# B&R Automation Studio project A2019059_Linka_Power_CP (part 27)

```iecst
        290:
            SC_P2_StoperSrobovania.StepName:='290 - Automaticky Rezim - modwel 5F presun manipulatora vzad';
            SC_P2_StoperSrobovania.IdleTime.PT:= T#200ms;
            SC_P2_StoperSrobovania.AlarmTime.PT:= T#5s;

            IF NOT SC_P2_StoperSrobovania.Switch1 AND P2_Robot.KOM_IN.Stav_RobotBezpPozicia_Srobovanie THEN
                P2_StoperSrobovania.OUT.KOM_PresunManipulator_DOZADU:= TRUE;
                SC_P2_StoperSrobovania.Switch1:= TRUE;
            END_IF

            IF P2_Srobovanie.OUT.KOM_PresunVZAD_Ukonceny THEN
                P2_Srobovanie.OUT.KOM_PresunVZAD_Ukonceny:= FALSE;
                P2_StoperSrobovania.OUT.KOM_PresunManipulator_DOZADU:= FALSE;
                CAM10.STAV.Results_READY:= FALSE;
                SC_P2_StoperSrobovania.ResetStep:= TRUE;
                SC_P2_StoperSrobovania.Step:= 293;
            END_IF

        293:
            SC_P2_StoperSrobovania.StepName:='293 - Automaticky Rezim - modwel 5F kamerova kontrola paletky CAM10';//CAM 10//
            SC_P2_StoperSrobovania.IdleTime.PT:= T#5s;
            SC_P2_StoperSrobovania.AlarmTime.PT:= T#5s;

            IF NOT SC_P2_StoperSrobovania.Switch1 AND CAM10.STAV.Command_READY THEN
                CAM10.CMD.Triger:= TRUE;
                SC_P2_StoperSrobovania.IdleTime.IN:= TRUE;
                SC_P2_StoperSrobovania.Switch1:= TRUE;
            END_IF

            IF CAM10.STAV.Results_READY AND CAM10.STAV.Command_AKCEPTOVANY THEN
                PocetTrigrovKamery:= 0;
                CAM10.STAV.Results_READY:= FALSE;
                SC_P2_StoperSrobovania.ResetStep:= TRUE;
                SC_P2_StoperSrobovania.Step:= 295;
            ELSIF SC_P2_StoperSrobovania.IdleTime.Q AND PocetTrigrovKamery < 5 THEN
                PocetTrigrovKamery:= PocetTrigrovKamery + 1;
                CAM10.STAV.Results_READY:= FALSE;
                CAM10.CMD.Triger:= FALSE;
                SC_P2_StoperSrobovania.ResetStep:= TRUE;
                SC_P2_StoperSrobovania.Step:= 294;
            ELSIF SC_P2_StoperSrobovania.IdleTime.Q AND PocetTrigrovKamery >= 5 THEN
                P2_Alarmy[295]:= TRUE;
                P2_PoruchaST3:= TRUE;
            END_IF

        294:
            SC_P2_StoperSrobovania.StepName:='294 - Automaticky Rezim - modwel 5F cakam na opatovny triger kamery';//CAM 10//
            SC_P2_StoperSrobovania.IdleTime.PT:= T#1s;
            SC_P2_StoperSrobovania.AlarmTime.PT:= T#5s;

            SC_P2_StoperSrobovania.IdleTime.IN:= TRUE;

            IF SC_P2_StoperSrobovania.IdleTime.Q THEN
                SC_P2_StoperSrobovania.ResetStep:= TRUE;
                SC_P2_StoperSrobovania.Step:= 293;
            END_IF

        295:
            SC_P2_StoperSrobovania.StepName:='295 - Automaticky Rezim - model 5F kontrola vysledku kamery';
            SC_P2_StoperSrobovania.IdleTime.PT:= T#200ms;
            SC_P2_StoperSrobovania.AlarmTime.PT:= T#5s;
            SC_P2_StoperSrobovania.IdleTime.IN:= TRUE;

            IF NOT CAM10.STAV.BUSY THEN
                CAM10.CMD.Triger:= FALSE;
				IF NOT CAM10.RESULT.Paletka.Pritomn_Busbarov_5F THEN
					CAM10.PAR.ResultFotky:= 'PASS';
					SC_P2_StoperSrobovania.ResetStep:= TRUE;
					SC_P2_StoperSrobovania.Step:= 300;
				ELSE
                    CAM10.PAR.ResultFotky:= 'FAIL';
                    SC_P2_StoperSrobovania.ResetStep:= TRUE;
                    SC_P2_StoperSrobovania.Step:= 300;
                END_IF
            END_IF

        300:
            SC_P2_StoperSrobovania.StepName:='300 - Automaticky Rezim - model 5F rozhodnutie podla kamerovej kontroly paletky';
            SC_P2_StoperSrobovania.IdleTime.PT:= T#200ms;
            SC_P2_StoperSrobovania.AlarmTime.PT:= T#5s;
            P2_Srobov_CakaNaKameru:= TRUE;

            IF CAM10.PAR.ResultFotky = 'PASS' THEN
                Paletka[i].PAR.StavPowerCP:= 'PASS';
                Paletka[i].VnutornyStav.CinnostUkoncena:= TRUE;
                P2_Srobov_CakaNaKameru:= FALSE;
                SC_P2_StoperSrobovania.ResetStep:= TRUE;
                SC_P2_StoperSrobovania.Step:= 540;
            ELSIF CAM10.PAR.ResultFotky = 'FAIL' THEN
                P2_Vizu.ZobrazHL2_ST5:= TRUE;
                Paletka[i].VnutornyStav.CinnostUkoncena:= TRUE;
                IF P2_Srobov_KAM_Result_OFF THEN
                    Paletka[i].PAR.StavPowerCP:= 'PASS';
                    P2_Vizu.ZobrazHL2_ST5:= FALSE;
                    P2_Srobov_CakaNaKameru:= FALSE;
                    SC_P2_StoperSrobovania.ResetStep:= TRUE;
                    SC_P2_StoperSrobovania.Step:= 540;
                ELSIF P2_Srobov_KAM_Result_OK THEN
                    P2_Srobov_KAM_Result_OK:= FALSE;
                    Paletka[i].PAR.StavPowerCP:= 'PASS';
                    CAM10.PAR.ResultFotky:= 'PASS';
                    P2_Srobov_CakaNaKameru:= FALSE;
                    P2_Vizu.ZobrazHL2_ST5:= FALSE;
                    SC_P2_StoperSrobovania.ResetStep:= TRUE;
                    SC_P2_StoperSrobovania.Step:= 540;
                ELSIF P2_Srobov_KAM_Result_NG THEN
                    P2_Srobov_KAM_Result_NG:= FALSE;
                    P2_Vizu.ZobrazHL2_ST5:= FALSE;
                    Paletka[i].PAR.StavPowerCP:= 'FAIL';
                    P2_Srobov_CakaNaKameru:= FALSE;
                    SC_P2_StoperSrobovania.ResetStep:= TRUE;
                    SC_P2_StoperSrobovania.Step:= 540;
                END_IF
            END_IF

            //********************************************Model 5H**************************************************************//

        358:
            SC_P2_StoperSrobovania.StepName:='358 - Automaticky Rezim - model 5H presun manipulatora vpred a odobratie vrchnych busbarov';
            SC_P2_StoperSrobovania.IdleTime.PT:= T#200ms;
            SC_P2_StoperSrobovania.AlarmTime.PT:= T#5s;

            P2_Robot.KOM_OUT.ManipSrobovania_BezpecnaPozicia:= TRUE;

            IF P2_Robot.KOM_IN.Stav_RobotBezpPozicia_Srobovanie AND NOT P2_Robot.KOM_IN.Stav_Busbary5H_Odobrate AND NOT P2_Robot.STAV.Zvaranie_PrebiehaManipulacia AND SC_P2_Srobovanie.Step = 100  THEN
                P2_StoperSrobovania.OUT.KOM_PresunManipulator_DOPREDU:= TRUE;
                P2_Robot.KOM_OUT.Odober_Busbary5H:= TRUE;
                Paletka[i].VnutornyStav.CinnostSpustena:= TRUE;
                SC_P2_StoperSrobovania.ResetStep:= TRUE;
                SC_P2_StoperSrobovania.Step:= 360;
            ELSIF NOT P2_Robot.KOM_IN.Stav_ProgramRUN THEN
                P2_Alarmy[271]:= TRUE;
                P2_PoruchaST3:= TRUE;
            END_IF

        360:
            SC_P2_StoperSrobovania.StepName:='360 - Automaticky Rezim - modwel 5H cakam na polozenie vrchnych busbarov';
            SC_P2_StoperSrobovania.IdleTime.PT:= T#200ms;
            SC_P2_StoperSrobovania.AlarmTime.PT:= T#5s;

            IF P2_Srobovanie.OUT.KOM_PresunVPRED_Ukonceny AND P2_Robot.KOM_IN.Stav_Busbary5H_Odobrate AND NOT P2_Robot.KOM_IN.Stav_Busbary5H_Polozene THEN
                P2_Srobovanie.OUT.KOM_PresunVPRED_Ukonceny:= FALSE;
                P2_StoperSrobovania.OUT.KOM_PresunManipulator_DOPREDU:= FALSE;
                P2_Robot.KOM_OUT.Odober_Busbary5H:= FALSE;
                SC_P2_StoperSrobovania.ResetStep:= TRUE;
                SC_P2_StoperSrobovania.Step:= 363;
            ELSIF NOT P2_Robot.KOM_IN.Stav_ProgramRUN THEN
                P2_Alarmy[271]:= TRUE;
                P2_PoruchaST3:= TRUE;
            END_IF

        363:
            SC_P2_StoperSrobovania.StepName:='363 - Automaticky Rezim - modwel 5H poloz vrchne busbary';
            SC_P2_StoperSrobovania.IdleTime.PT:= T#200ms;
            SC_P2_StoperSrobovania.AlarmTime.PT:= T#5s;

            P2_Robot.KOM_OUT.ManipSrobovania_BezpecnaPozicia:= TRUE;

            IF NOT SC_P2_StoperSrobovania.Switch1 AND NOT P2_Robot.KOM_IN.Stav_Busbary5H_Odobrate THEN
                P2_Robot.KOM_OUT.Poloz_Busbary5H:= TRUE;
                SC_P2_StoperSrobovania.Switch1:= TRUE;
            END_IF

            IF P2_Robot.KOM_IN.Stav_Busbary5H_Polozene THEN
                P2_Robot.KOM_OUT.Poloz_Busbary5H:= FALSE;
                SC_P2_StoperSrobovania.ResetStep:= TRUE;
                SC_P2_StoperSrobovania.Step:= 365;
            ELSIF NOT P2_Robot.KOM_IN.Stav_ProgramRUN THEN
                P2_Alarmy[271]:= TRUE;
                P2_PoruchaST3:= TRUE;
            END_IF

        365:
            SC_P2_StoperSrobovania.StepName:='365 - Automaticky Rezim - modwel 5H zaskrutkuj skrutku M4';
            SC_P2_StoperSrobovania.IdleTime.PT:= T#200ms;
            SC_P2_StoperSrobovania.AlarmTime.PT:= T#5s;

            IF NOT SC_P2_StoperSrobovania.Switch1 THEN
                P2_Srobovanie.STAV.Vysledok_Srobovania:= '';
                P2_StoperSrobovania.OUT.KOM_5H_ZasrobujSkrutkuM4:= TRUE;
                SC_P2_StoperSrobovania.Switch1:= TRUE;
            END_IF

            IF P2_Srobovanie.OUT.KOM_Srobovanie_Ukoncene AND NOT P2_Robot.KOM_IN.Stav_Filter5H_Dotlaceny THEN
                P2_Srobovanie.OUT.KOM_Srobovanie_Ukoncene:= FALSE;
                P2_StoperSrobovania.OUT.KOM_5H_ZasrobujSkrutkuM4:= FALSE;
                IF P2_StoperSrobovania.STAV.Porucha THEN
                    SC_P2_StoperSrobovania.ResetStep:= TRUE;
                    SC_P2_StoperSrobovania.Step:= 500;//500
                ELSE
                    SC_P2_StoperSrobovania.ResetStep:= TRUE;
                    SC_P2_StoperSrobovania.Step:= 368;
                END_IF
            END_IF

        368:
            SC_P2_StoperSrobovania.StepName:='368 - Automaticky Rezim - modwel 5H kontrola vysledku zaskrutkovania skrutky M4';
            SC_P2_StoperSrobovania.IdleTime.PT:= T#200ms;
            SC_P2_StoperSrobovania.AlarmTime.PT:= T#5s;

            Reports.Skrutkovacky.Moment_ToleranciaMIN.P2_StrednaSkrutkaM4:= REAL_TO_STRING(P2_Srobovanie.STAV.M4_Moment_ToleranciaMIN_REAL);
            Reports.Skrutkovacky.Moment_ToleranciaMAX.P2_StrednaSkrutkaM4:= REAL_TO_STRING(P2_Srobovanie.STAV.M4_Moment_ToleranciaMAX_REAL);
            Reports.Skrutkovacky.Moment_NameranaHodnota.P2_StrednaSkrutkaM4:= REAL_TO_STRING(P2_Srobovanie.STAV.M4_DosiahnutyMoment_REAL);
            Reports.Skrutkovacky.Uhol_ToleranciaMIN.P2_StrednaSkrutkaM4:= UDINT_TO_STRING(P2_Srobovanie.STAV.M4_Uhol_ToleranciaMIN);
            Reports.Skrutkovacky.Uhol_ToleranciaMAX.P2_StrednaSkrutkaM4:= UDINT_TO_STRING(P2_Srobovanie.STAV.M4_Uhol_ToleranciaMAX);
            Reports.Skrutkovacky.Uhol_NameranaHodnota.P2_StrednaSkrutkaM4:= UDINT_TO_STRING(P2_Srobovanie.STAV.M4_DosiahnutyUhol);

            IF NOT SC_P2_StoperSrobovania.Switch1 THEN
                P2_Skrutk_5H_StrednaM4_Vysunutie:= STRING_TO_REAL(Reports.Skrutkovacky.VyskaSkrutkovania.P2_StrednaSkrutkaM4);
                IF (P2_Skrutk_5H_StrednaM4_Vysunutie <= P2_RemPremenne.P2_Srob5H_StrednaM4_Vysunutie_HI) AND (P2_Skrutk_5H_StrednaM4_Vysunutie >= P2_RemPremenne.P2_Srob5H_StrednaM4_Vysunutie_LO)THEN
                    VysunutieSkrutkovacky_OK:= TRUE;
                ELSE
                    VysunutieSkrutkovacky_OK:= FALSE;
                END_IF
                SC_P2_StoperSrobovania.Switch1:= TRUE;
            END_IF

            IF P2_Srobovanie.STAV.Vysledok_Srobovania = 'OK' THEN
                IF VysunutieSkrutkovacky_OK THEN
                    Reports.Skrutkovacky.VyslednyReport.P2_StrednaSkrutkaM4:= 'PASS';
                    SC_P2_StoperSrobovania.ResetStep:= TRUE;
                    SC_P2_StoperSrobovania.Step:= 370;
                ELSE
                    Reports.Skrutkovacky.VyslednyReport.P2_StrednaSkrutkaM4:= 'FAIL';
                    IF P2_Srobov_M4_Result_OFF THEN
                        SC_P2_StoperSrobovania.ResetStep:= TRUE;
                        SC_P2_StoperSrobovania.Step:= 370;
                    ELSE
                        DoskrutkovaniePriPoruche:= TRUE;
                        SC_P2_StoperSrobovania.ResetStep:= TRUE;
                        SC_P2_StoperSrobovania.Step:= 370;//500
                    END_IF
                END_IF
            ELSIF P2_Srobovanie.STAV.Vysledok_Srobovania = 'NG' THEN
                Reports.Skrutkovacky.VyslednyReport.P2_StrednaSkrutkaM4:= 'FAIL';
                IF P2_Srobov_M4_Result_OFF THEN
                    SC_P2_StoperSrobovania.ResetStep:= TRUE;
                    SC_P2_StoperSrobovania.Step:= 370;
                ELSE
                    DoskrutkovaniePriPoruche:= TRUE;
                    SC_P2_StoperSrobovania.ResetStep:= TRUE;
                    SC_P2_StoperSrobovania.Step:= 370;//500
                END_IF
            END_IF

        370:
            SC_P2_StoperSrobovania.StepName:='370 - Automaticky Rezim - modwel 5H dotlac filter';
            SC_P2_StoperSrobovania.IdleTime.PT:= T#200ms;
            SC_P2_StoperSrobovania.AlarmTime.PT:= T#5s;

            P2_Robot.KOM_OUT.ManipSrobovania_BezpecnaPozicia:= TRUE;

            IF NOT SC_P2_StoperSrobovania.Switch1 THEN
                P2_Robot.KOM_OUT.Dotlac_Filter5H:= TRUE;
                SC_P2_StoperSrobovania.Switch1:= TRUE;
            END_IF

            IF P2_Robot.KOM_IN.Stav_Filter5H_Dotlaceny THEN
                P2_Robot.KOM_OUT.Dotlac_Filter5H:= FALSE;
                SC_P2_StoperSrobovania.ResetStep:= TRUE;
                SC_P2_StoperSrobovania.Step:= 375;
            ELSIF NOT P2_Robot.KOM_IN.Stav_ProgramRUN THEN
                P2_Alarmy[271]:= TRUE;
                P2_PoruchaST3:= TRUE;
            END_IF

        375:
            SC_P2_StoperSrobovania.StepName:='375 - Automaticky Rezim - modwel 5H zaskrutkuj lavu skrutku M5';
            SC_P2_StoperSrobovania.IdleTime.PT:= T#200ms;
            SC_P2_StoperSrobovania.AlarmTime.PT:= T#5s;

            IF NOT SC_P2_StoperSrobovania.Switch1 THEN
                P2_Srobovanie.STAV.Vysledok_Srobovania:= '';
                P2_StoperSrobovania.OUT.KOM_5H_ZasrobujLavuSkrutkuM5:= TRUE;
                SC_P2_StoperSrobovania.Switch1:= TRUE;
            END_IF

            IF P2_Srobovanie.OUT.KOM_Srobovanie_Ukoncene THEN
                P2_Srobovanie.OUT.KOM_Srobovanie_Ukoncene:= FALSE;
                P2_StoperSrobovania.OUT.KOM_5H_ZasrobujLavuSkrutkuM5:= FALSE;
                IF P2_StoperSrobovania.STAV.Porucha THEN
                    SC_P2_StoperSrobovania.ResetStep:= TRUE;
                    SC_P2_StoperSrobovania.Step:= 500;
                ELSE
                    SC_P2_StoperSrobovania.ResetStep:= TRUE;
                    SC_P2_StoperSrobovania.Step:= 378;
                END_IF
            END_IF

        378:
            SC_P2_StoperSrobovania.StepName:='378 - Automaticky Rezim - modwel 5H kontrola vysledku zaskrutkovania lavej skrutky M5';
            SC_P2_StoperSrobovania.IdleTime.PT:= T#200ms;
            SC_P2_StoperSrobovania.AlarmTime.PT:= T#5s;

            Reports.Skrutkovacky.Moment_ToleranciaMIN.P2_LavaSkrutkaM5:= REAL_TO_STRING(P2_Srobovanie.STAV.M5_Moment_ToleranciaMIN_REAL);
            Reports.Skrutkovacky.Moment_ToleranciaMAX.P2_LavaSkrutkaM5:= REAL_TO_STRING(P2_Srobovanie.STAV.M5_Moment_ToleranciaMAX_REAL);
            Reports.Skrutkovacky.Moment_NameranaHodnota.P2_LavaSkrutkaM5:= REAL_TO_STRING(P2_Srobovanie.STAV.M5_DosiahnutyMoment_REAL);
            Reports.Skrutkovacky.Uhol_ToleranciaMIN.P2_LavaSkrutkaM5:= UDINT_TO_STRING(P2_Srobovanie.STAV.M5_Uhol_ToleranciaMIN);
            Reports.Skrutkovacky.Uhol_ToleranciaMAX.P2_LavaSkrutkaM5:= UDINT_TO_STRING(P2_Srobovanie.STAV.M5_Uhol_ToleranciaMAX);
            Reports.Skrutkovacky.Uhol_NameranaHodnota.P2_LavaSkrutkaM5:= UDINT_TO_STRING(P2_Srobovanie.STAV.M5_DosiahnutyUhol);

            IF NOT SC_P2_StoperSrobovania.Switch1 THEN
                P2_Skrutk_5H_LavaM5_Vysunutie:= STRING_TO_REAL(Reports.Skrutkovacky.VyskaSkrutkovania.P2_LavaSkrutkaM5);
                IF (P2_Skrutk_5H_LavaM5_Vysunutie <= P2_RemPremenne.P2_Srob5H_LavaM5_Vysunutie_HI) AND (P2_Skrutk_5H_LavaM5_Vysunutie >= P2_RemPremenne.P2_Srob5H_LavaM5_Vysunutie_LO)THEN
                    VysunutieSkrutkovacky_OK:= TRUE;
                ELSE
                    VysunutieSkrutkovacky_OK:= FALSE;
                END_IF
                SC_P2_StoperSrobovania.Switch1:= TRUE;
            END_IF

            IF P2_Srobovanie.STAV.Vysledok_Srobovania = 'OK' THEN
                IF VysunutieSkrutkovacky_OK THEN
                    IF NOT DoskrutkovaniePriPoruche THEN
                        Reports.Skrutkovacky.VyslednyReport.P2_LavaSkrutkaM5:= 'PASS';
                    ELSE
                        Reports.Skrutkovacky.VyslednyReport.P2_LavaSkrutkaM5:= 'FAIL';
                    END_IF
                    SC_P2_StoperSrobovania.ResetStep:= TRUE;
                    SC_P2_StoperSrobovania.Step:= 380;
                ELSE
                    Reports.Skrutkovacky.VyslednyReport.P2_LavaSkrutkaM5:= 'FAIL';
                    IF P2_Srobov_M5_Result_OFF THEN
                        SC_P2_StoperSrobovania.ResetStep:= TRUE;
                        SC_P2_StoperSrobovania.Step:= 380;
                    ELSE
                        DoskrutkovaniePriPoruche:= TRUE;
                        SC_P2_StoperSrobovania.ResetStep:= TRUE;
                        SC_P2_StoperSrobovania.Step:= 380;//500
                    END_IF
                END_IF
            ELSIF P2_Srobovanie.STAV.Vysledok_Srobovania = 'NG' THEN
                Reports.Skrutkovacky.VyslednyReport.P2_LavaSkrutkaM5:= 'FAIL';
                IF P2_Srobov_M5_Result_OFF THEN
                    SC_P2_StoperSrobovania.ResetStep:= TRUE;
                    SC_P2_StoperSrobovania.Step:= 380;
                ELSE
                    DoskrutkovaniePriPoruche:= TRUE;
                    SC_P2_StoperSrobovania.ResetStep:= TRUE;
                    SC_P2_StoperSrobovania.Step:= 380;//500
                END_IF
            END_IF

        380:
            SC_P2_StoperSrobovania.StepName:='380 - Automaticky Rezim - modwel 5H zaskrutkuj pravu skrutku M5';
            SC_P2_StoperSrobovania.IdleTime.PT:= T#200ms;
            SC_P2_StoperSrobovania.AlarmTime.PT:= T#5s;

            IF NOT SC_P2_StoperSrobovania.Switch1  THEN
                P2_Srobovanie.STAV.Vysledok_Srobovania:= '';
                P2_StoperSrobovania.OUT.KOM_5H_ZasrobujPravuSkrutkuM5:= TRUE;
                SC_P2_StoperSrobovania.Switch1:= TRUE;
            END_IF

            IF P2_Srobovanie.OUT.KOM_Srobovanie_Ukoncene THEN
                P2_Srobovanie.OUT.KOM_Srobovanie_Ukoncene:= FALSE;
                P2_StoperSrobovania.OUT.KOM_5H_ZasrobujPravuSkrutkuM5:= FALSE;
                IF P2_StoperSrobovania.STAV.Porucha THEN
                    SC_P2_StoperSrobovania.ResetStep:= TRUE;
                    SC_P2_StoperSrobovania.Step:= 500;
                ELSE
                    SC_P2_StoperSrobovania.ResetStep:= TRUE;
                    SC_P2_StoperSrobovania.Step:= 383;
                END_IF
            END_IF

        383:
            SC_P2_StoperSrobovania.StepName:='383 - Automaticky Rezim - modwel 5H kontrola vysledku zaskrutkovania pravej skrutky M5';
            SC_P2_StoperSrobovania.IdleTime.PT:= T#200ms;
            SC_P2_StoperSrobovania.AlarmTime.PT:= T#5s;

            Reports.Skrutkovacky.Moment_ToleranciaMIN.P2_PravaSkrutkaM5:= REAL_TO_STRING(P2_Srobovanie.STAV.M5_Moment_ToleranciaMIN_REAL);
            Reports.Skrutkovacky.Moment_ToleranciaMAX.P2_PravaSkrutkaM5:= REAL_TO_STRING(P2_Srobovanie.STAV.M5_Moment_ToleranciaMAX_REAL);
            Reports.Skrutkovacky.Moment_NameranaHodnota.P2_PravaSkrutkaM5:= REAL_TO_STRING(P2_Srobovanie.STAV.M5_DosiahnutyMoment_REAL);
            Reports.Skrutkovacky.Uhol_ToleranciaMIN.P2_PravaSkrutkaM5:= UDINT_TO_STRING(P2_Srobovanie.STAV.M5_Uhol_ToleranciaMIN);
            Reports.Skrutkovacky.Uhol_ToleranciaMAX.P2_PravaSkrutkaM5:= UDINT_TO_STRING(P2_Srobovanie.STAV.M5_Uhol_ToleranciaMAX);
            Reports.Skrutkovacky.Uhol_NameranaHodnota.P2_PravaSkrutkaM5:= UDINT_TO_STRING(P2_Srobovanie.STAV.M5_DosiahnutyUhol);

            IF NOT SC_P2_StoperSrobovania.Switch1 THEN
                P2_Skrutk_5H_PravaM5_Vysunutie:= STRING_TO_REAL(Reports.Skrutkovacky.VyskaSkrutkovania.P2_PravaSkrutkaM5);
                IF (P2_Skrutk_5H_PravaM5_Vysunutie <= P2_RemPremenne.P2_Srob5H_PravaM5_Vysunutie_HI) AND (P2_Skrutk_5H_PravaM5_Vysunutie >= P2_RemPremenne.P2_Srob5H_PravaM5_Vysunutie_LO)THEN
                    VysunutieSkrutkovacky_OK:= TRUE;
                ELSE
                    VysunutieSkrutkovacky_OK:= FALSE;
                END_IF
                SC_P2_StoperSrobovania.Switch1:= TRUE;
            END_IF

            IF P2_Srobovanie.STAV.Vysledok_Srobovania = 'OK' THEN
                IF VysunutieSkrutkovacky_OK THEN
                    IF NOT DoskrutkovaniePriPoruche THEN
                        Reports.Skrutkovacky.VyslednyReport.P2_PravaSkrutkaM5:= 'PASS';
                        SC_P2_StoperSrobovania.ResetStep:= TRUE;
                        SC_P2_StoperSrobovania.Step:= 385;
                    ELSE
                        Reports.Skrutkovacky.VyslednyReport.P2_PravaSkrutkaM5:= 'FAIL';
                        SC_P2_StoperSrobovania.ResetStep:= TRUE;
                        SC_P2_StoperSrobovania.Step:= 500;
                    END_IF
                ELSE
                    Reports.Skrutkovacky.VyslednyReport.P2_PravaSkrutkaM5:= 'FAIL';
                    IF P2_Srobov_M5_Result_OFF THEN
                        SC_P2_StoperSrobovania.ResetStep:= TRUE;
                        SC_P2_StoperSrobovania.Step:= 385;
                    ELSE
                        SC_P2_StoperSrobovania.ResetStep:= TRUE;
                        SC_P2_StoperSrobovania.Step:= 500;
                    END_IF
                END_IF
            ELSIF P2_Srobovanie.STAV.Vysledok_Srobovania = 'NG' THEN
                Reports.Skrutkovacky.VyslednyReport.P2_PravaSkrutkaM5:= 'FAIL';
                IF P2_Srobov_M5_Result_OFF THEN
                    SC_P2_StoperSrobovania.ResetStep:= TRUE;
                    SC_P2_StoperSrobovania.Step:= 385;
                ELSE
                    SC_P2_StoperSrobovania.ResetStep:= TRUE;
                    SC_P2_StoperSrobovania.Step:= 500;
                END_IF
            END_IF

        385:
            SC_P2_StoperSrobovania.StepName:='385 - Automaticky Rezim - modwel 5H presun manipulatora vpred, vystavenie signalu pre robota chod do cakacej pozicie ';
            SC_P2_StoperSrobovania.IdleTime.PT:= T#200ms;
            SC_P2_StoperSrobovania.AlarmTime.PT:= T#5s;

            P2_Robot.KOM_OUT.ManipSrobovania_BezpecnaPozicia:= TRUE;

            IF NOT P2_Robot.KOM_IN.Stav_RobotPoziciaCakania THEN
                P2_StoperSrobovania.OUT.KOM_PresunManipulator_DOPREDU:= TRUE;
                P2_Robot.KOM_OUT.Presun_CakaciaPozicia:= TRUE;
                SC_P2_StoperSrobovania.ResetStep:= TRUE;
                SC_P2_StoperSrobovania.Step:= 388;
            END_IF

        388:
            SC_P2_StoperSrobovania.StepName:='388 - Automaticky Rezim - model 5H cakam na presunutie robota do cakacej pozicie';
            SC_P2_StoperSrobovania.IdleTime.PT:= T#200ms;
            SC_P2_StoperSrobovania.AlarmTime.PT:= T#5s;

            IF P2_Srobovanie.OUT.KOM_PresunVPRED_Ukonceny AND P2_Robot.KOM_IN.Stav_RobotPoziciaCakania THEN
                P2_Robot.KOM_OUT.Presun_CakaciaPozicia:= FALSE;
                P2_Robot.STAV.Srobovanie_PrebiehaManipulacia:= FALSE;
                P2_Srobovanie.OUT.KOM_PresunVPRED_Ukonceny:= FALSE;
                P2_StoperSrobovania.OUT.KOM_PresunManipulator_DOPREDU:= FALSE;
                SC_P2_StoperSrobovania.ResetStep:= TRUE;
                SC_P2_StoperSrobovania.Step:= 390;
            END_IF

        390:
            SC_P2_StoperSrobovania.StepName:='390 - Automaticky Rezim - modwel 5H presun manipulatora vzad';
            SC_P2_StoperSrobovania.IdleTime.PT:= T#200ms;
            SC_P2_StoperSrobovania.AlarmTime.PT:= T#5s;

            IF NOT SC_P2_StoperSrobovania.Switch1 AND P2_Robot.KOM_IN.Stav_RobotBezpPozicia_Srobovanie AND SC_P2_Srobovanie.Step = 100 THEN
                P2_StoperSrobovania.OUT.KOM_PresunManipulator_DOZADU:= TRUE;
                SC_P2_StoperSrobovania.Switch1:= TRUE;
            END_IF

            IF P2_Srobovanie.OUT.KOM_PresunVZAD_Ukonceny THEN
                P2_Srobovanie.OUT.KOM_PresunVZAD_Ukonceny:= FALSE;
                P2_StoperSrobovania.OUT.KOM_PresunManipulator_DOZADU:= FALSE;
                CAM10.STAV.Results_READY:= FALSE;
                SC_P2_StoperSrobovania.ResetStep:= TRUE;
                SC_P2_StoperSrobovania.Step:= 393;
            END_IF

        393:
            SC_P2_StoperSrobovania.StepName:='393 - Automaticky Rezim - modwel 5H kamerova kontrola paletky CAM10';//CAM 10//
            SC_P2_StoperSrobovania.IdleTime.PT:= T#5s;
            SC_P2_StoperSrobovania.AlarmTime.PT:= T#5s;

            IF NOT SC_P2_StoperSrobovania.Switch1 AND CAM10.STAV.Command_READY THEN
                CAM10.CMD.Triger:= TRUE;
                SC_P2_StoperSrobovania.IdleTime.IN:= TRUE;
                SC_P2_StoperSrobovania.Switch1:= TRUE;
            END_IF

            IF CAM10.STAV.Results_READY AND CAM10.STAV.Command_AKCEPTOVANY THEN
                PocetTrigrovKamery:= 0;
                CAM10.STAV.Results_READY:= FALSE;
                SC_P2_StoperSrobovania.ResetStep:= TRUE;
                SC_P2_StoperSrobovania.Step:= 395;
            ELSIF SC_P2_StoperSrobovania.IdleTime.Q AND PocetTrigrovKamery < 5 THEN
                PocetTrigrovKamery:= PocetTrigrovKamery + 1;
                CAM10.STAV.Results_READY:= FALSE;
                CAM10.CMD.Triger:= FALSE;
                SC_P2_StoperSrobovania.ResetStep:= TRUE;
                SC_P2_StoperSrobovania.Step:= 394;
            ELSIF SC_P2_StoperSrobovania.IdleTime.Q AND PocetTrigrovKamery >= 5 THEN
                P2_Alarmy[295]:= TRUE;
                P2_PoruchaST3:= TRUE;
            END_IF

        394:
            SC_P2_StoperSrobovania.StepName:='394 - Automaticky Rezim - modwel 5H cakam na opatovny triger kamery';//CAM 10//
            SC_P2_StoperSrobovania.IdleTime.PT:= T#1s;
            SC_P2_StoperSrobovania.AlarmTime.PT:= T#5s;

            SC_P2_StoperSrobovania.IdleTime.IN:= TRUE;

            IF SC_P2_StoperSrobovania.IdleTime.Q THEN
                SC_P2_StoperSrobovania.ResetStep:= TRUE;
                SC_P2_StoperSrobovania.Step:= 393;
            END_IF

        395:
            SC_P2_StoperSrobovania.StepName:='395 - Automaticky Rezim - model 5H kontrola vysledku kamery';
            SC_P2_StoperSrobovania.IdleTime.PT:= T#200ms;
            SC_P2_StoperSrobovania.AlarmTime.PT:= T#5s;
            SC_P2_StoperSrobovania.IdleTime.IN:= TRUE;

            IF NOT CAM10.STAV.BUSY  THEN
                CAM10.CMD.Triger:= FALSE;
				IF NOT CAM10.RESULT.Paletka.Pritomn_Busbarov_5H THEN
					CAM10.PAR.ResultFotky:= 'PASS';
					SC_P2_StoperSrobovania.ResetStep:= TRUE;
					SC_P2_StoperSrobovania.Step:= 400;
                ELSE
                    CAM10.PAR.ResultFotky:= 'FAIL';
                    SC_P2_StoperSrobovania.ResetStep:= TRUE;
                    SC_P2_StoperSrobovania.Step:= 400;
                END_IF
            END_IF

        400:
            SC_P2_StoperSrobovania.StepName:='400 - Automaticky Rezim - model 5H rozhodnutie podla kamerovej kontroly paletky';
            SC_P2_StoperSrobovania.IdleTime.PT:= T#200ms;
            SC_P2_StoperSrobovania.AlarmTime.PT:= T#5s;
            P2_Srobov_CakaNaKameru:= TRUE;

            IF CAM10.PAR.ResultFotky = 'PASS' THEN
                Paletka[i].VnutornyStav.CinnostUkoncena:= TRUE;
                Paletka[i].PAR.StavPowerCP:= 'PASS';
                P2_Srobov_CakaNaKameru:= FALSE;
                SC_P2_StoperSrobovania.ResetStep:= TRUE;
                SC_P2_StoperSrobovania.Step:= 540;
            ELSIF CAM10.PAR.ResultFotky = 'FAIL' THEN
                P2_Vizu.ZobrazHL3_ST5:= TRUE;
                Paletka[i].VnutornyStav.CinnostUkoncena:= TRUE;
                IF P2_Srobov_KAM_Result_OFF THEN
                    Paletka[i].PAR.StavPowerCP:= 'PASS';
                    P2_Vizu.ZobrazHL3_ST5:= FALSE;
                    P2_Srobov_CakaNaKameru:= FALSE;
                    SC_P2_StoperSrobovania.ResetStep:= TRUE;
                    SC_P2_StoperSrobovania.Step:= 540;
                ELSIF P2_Srobov_KAM_Result_OK THEN
                    P2_Srobov_KAM_Result_OK:= FALSE;
                    Paletka[i].PAR.StavPowerCP:= 'PASS';
                    CAM10.PAR.ResultFotky:= 'PASS';
                    P2_Srobov_CakaNaKameru:= FALSE;
                    P2_Vizu.ZobrazHL3_ST5:= FALSE;
                    SC_P2_StoperSrobovania.ResetStep:= TRUE;
                    SC_P2_StoperSrobovania.Step:= 540;
                ELSIF P2_Srobov_KAM_Result_NG THEN
                    P2_Srobov_KAM_Result_NG:= FALSE;
                    P2_Vizu.ZobrazHL3_ST5:= FALSE;
                    Paletka[i].PAR.StavPowerCP:= 'FAIL';
                    P2_Srobov_CakaNaKameru:= FALSE;
                    SC_P2_StoperSrobovania.ResetStep:= TRUE;
                    SC_P2_StoperSrobovania.Step:= 540;
                END_IF
            END_IF

            //****************************************Uvolnenie robota a vyfotenie paletky po zlom skrutkovaní************************************************//

        500:
            SC_P2_StoperSrobovania.StepName:='500 - Automaticky Rezim - presun manipulatora vpred';
            SC_P2_StoperSrobovania.IdleTime.PT:= T#200ms;
            SC_P2_StoperSrobovania.AlarmTime.PT:= T#5s;

			Paletka[i].PAR.StavPaletky:= 'NG';

            IF NOT SC_P2_StoperSrobovania.Switch1 THEN
                P2_StoperSrobovania.OUT.KOM_PresunManipulator_DOPREDU:= TRUE;
                SC_P2_StoperSrobovania.Switch1:= TRUE;
            END_IF

            IF P2_Srobovanie.OUT.KOM_PresunVPRED_Ukonceny THEN
                P2_Srobovanie.OUT.KOM_PresunVPRED_Ukonceny:= FALSE;
                P2_StoperSrobovania.OUT.KOM_PresunManipulator_DOPREDU:= FALSE;
                SC_P2_StoperSrobovania.ResetStep:= TRUE;
                SC_P2_StoperSrobovania.Step:= 503;
            END_IF

        503:
            SC_P2_StoperSrobovania.StepName:='503 - Automaticky Rezim - vystavenie signalu pre robota chod do cakacej pozicie';
            SC_P2_StoperSrobovania.IdleTime.PT:= T#200ms;
            SC_P2_StoperSrobovania.AlarmTime.PT:= T#5s;

            P2_Robot.KOM_OUT.ManipSrobovania_BezpecnaPozicia:= TRUE;

            IF NOT SC_P2_StoperSrobovania.Switch1 THEN
                P2_Robot.KOM_OUT.Presun_CakaciaPozicia:= TRUE;
                SC_P2_StoperSrobovania.Switch1:= TRUE;
            END_IF

            IF P2_Robot.KOM_IN.Stav_RobotBezpPozicia_Srobovanie THEN
                P2_Robot.KOM_OUT.Presun_CakaciaPozicia:= FALSE;
                SC_P2_StoperSrobovania.ResetStep:= TRUE;
                SC_P2_StoperSrobovania.Step:= 505;
            END_IF

        505:
            SC_P2_StoperSrobovania.StepName:='505 - Automaticky Rezim - presun manipulatora vzad';
            SC_P2_StoperSrobovania.IdleTime.PT:= T#200ms;
            SC_P2_StoperSrobovania.AlarmTime.PT:= T#5s;

            IF NOT SC_P2_StoperSrobovania.Switch1 THEN
                P2_StoperSrobovania.OUT.KOM_PresunManipulator_DOZADU:= TRUE;
                SC_P2_StoperSrobovania.Switch1:= TRUE;
            END_IF

            IF P2_Srobovanie.OUT.KOM_PresunVZAD_Ukonceny THEN
                P2_Srobovanie.OUT.KOM_PresunVZAD_Ukonceny:= FALSE;
                P2_StoperSrobovania.OUT.KOM_PresunManipulator_DOZADU:= FALSE;
                IF P2_StoperSrobovania.STAV.Porucha THEN
                    CAM10.STAV.Results_READY:= FALSE;
                    SC_P2_StoperSrobovania.ResetStep:= TRUE;
                    SC_P2_StoperSrobovania.Step:= 545;
                ELSE
                    SC_P2_StoperSrobovania.ResetStep:= TRUE;
                    SC_P2_StoperSrobovania.Step:= 508;
                END_IF
            END_IF

        508:
            SC_P2_StoperSrobovania.StepName:='508 - Automaticky Rezim - kamerova kontrola paletky CAM10';//CAM 10//
            SC_P2_StoperSrobovania.IdleTime.PT:= T#5s;
            SC_P2_StoperSrobovania.AlarmTime.PT:= T#5s;
            SC_P2_StoperSrobovania.IdleTime.IN:= TRUE;

            IF NOT SC_P2_StoperSrobovania.Switch1 AND CAM10.STAV.Command_READY THEN
                CAM10.CMD.Triger:= TRUE;
                SC_P2_StoperSrobovania.Switch1:= TRUE;
            END_IF

            IF CAM10.STAV.Results_READY AND CAM10.STAV.Command_AKCEPTOVANY THEN
                PocetTrigrovKamery:= 0;
                CAM10.STAV.Results_READY:= FALSE;
                Paletka[i].PAR.StavPowerCP:= 'FAIL';
                CAM10.PAR.ResultFotky:= 'FAIL';
                SC_P2_StoperSrobovania.ResetStep:= TRUE;
                SC_P2_StoperSrobovania.Step:= 540;
            ELSIF SC_P2_StoperSrobovania.IdleTime.Q AND PocetTrigrovKamery < 5 THEN
                PocetTrigrovKamery:= PocetTrigrovKamery + 1;
                CAM10.STAV.Results_READY:= FALSE;
                CAM10.CMD.Triger:= FALSE;
                SC_P2_StoperSrobovania.ResetStep:= TRUE;
                SC_P2_StoperSrobovania.Step:= 510;
            ELSIF SC_P2_StoperSrobovania.IdleTime.Q AND PocetTrigrovKamery >= 5 THEN
                P2_Alarmy[295]:= TRUE;
                P2_PoruchaST3:= TRUE;
            END_IF

        510:
            SC_P2_StoperSrobovania.StepName:='510 - Automaticky Rezim - cakam na opatovny triger kamery';//CAM 10//
            SC_P2_StoperSrobovania.IdleTime.PT:= T#1s;
            SC_P2_StoperSrobovania.AlarmTime.PT:= T#5s;

            SC_P2_StoperSrobovania.IdleTime.IN:= TRUE;

            IF SC_P2_StoperSrobovania.IdleTime.Q THEN
                SC_P2_StoperSrobovania.ResetStep:= TRUE;
                SC_P2_StoperSrobovania.Step:= 508;
            END_IF

            //Odoslanie fotiek na server//

        540:
            SC_P2_StoperSrobovania.StepName:='540 - Automaticky Rezim - odoslanie fotiek na server';
            SC_P2_StoperSrobovania.IdleTime.PT:= T#200ms;
            SC_P2_StoperSrobovania.AlarmTime.PT:= T#5s;

            IF NOT SC_P2_StoperSrobovania.Switch1 THEN
                FTP_CAM10.INPUTS.QRkodPowerCP:= Paletka[i].PAR.QRkodPowerCP;
                CisloFotky:= CisloFotky + 1;
                FTP_CAM10.INPUTS.IndexFotky:= USINT_TO_STRING(CisloFotky);
                FTP_CAM10.INPUTS.Result:= CAM6.PAR.ResultFotky;
                Reports.Kamery.P2_CAM10_KontrolaPaletky:= CAM10.PAR.ResultFotky;

                FTP_CAM10.CMD.OdosliFotku:= TRUE;
                SC_P2_StoperSrobovania.Switch1:= TRUE;
            END_IF

            IF FTP_CAM10.STATUS.KomunikaciaUkoncena THEN
                FTP_CAM10.CMD.OdosliFotku:= FALSE;
                Paletka[i].VnutornyStav.FotkyOdoslane:= TRUE;
                SC_P2_StoperSrobovania.ResetStep:= TRUE;
                SC_P2_StoperSrobovania.Step:= 545;
            ELSIF FTP_CAM10.STATUS.KomunikaciaError THEN
                P2_Alarmy[232]:= TRUE;
                P2_PoruchaST3:= TRUE;
            END_IF

            //Odcentrovanie paletky//
        545:
            SC_P2_StoperSrobovania.StepName:='545 - Automaticky Rezim - odcentrovanie paletky';
            SC_P2_StoperSrobovania.IdleTime.PT:= T#200ms;
            SC_P2_StoperSrobovania.AlarmTime.PT:= T#5s;

            IF NOT SC_P2_StoperSrobovania.Switch1 THEN
                Centrovacku_ZASUN:= TRUE;
                SC_P2_StoperSrobovania.Switch1:= TRUE;
            END_IF

            IF P2_StoperSrobovania.IN.Centrovanie_ZASUNUTE_IS15 THEN
                IF P2_StoperSrobovania.STAV.Porucha THEN
                    P2_PoruchaST3:= TRUE;
                ELSE
                    SC_P2_StoperSrobovania.ResetStep:= TRUE;
                    SC_P2_StoperSrobovania.Step:= 550;
                END_IF
            END_IF

            //Odoslanie dát na server//

        550:
            SC_P2_StoperSrobovania.StepName:='550 - Automaticky Rezim - odoslanie stavu paletky na server';
            SC_P2_StoperSrobovania.IdleTime.PT:= T#200ms;
            SC_P2_StoperSrobovania.AlarmTime.PT:= T#10s;

            IF NOT SC_P2_StoperSrobovania.Switch1 THEN
                TRCB_P2_Srobovanie_ST5.CMD.OdosliStavPaletky_TYP2:= TRUE;
                SC_P2_StoperSrobovania.Switch1:= TRUE;
            END_IF

            IF TRCB_P2_Srobovanie_ST5.STATUS.KomunikaciaUkoncena THEN
                TRCB_P2_Srobovanie_ST5.CMD.OdosliStavPaletky_TYP2:= FALSE;
                SC_P2_StoperSrobovania.ResetStep:= TRUE;
                SC_P2_StoperSrobovania.Step:= 553;
            ELSIF TRCB_P2_Srobovanie_ST5.STATUS.KomunikaciaError THEN
                //                P2_Alarmy[233]:= TRUE;
                //                P2_PoruchaST3:= TRUE;
            END_IF

        553:
            SC_P2_StoperSrobovania.StepName:='553 - Automaticky Rezim - kontrola odpovede servera';
            SC_P2_StoperSrobovania.IdleTime.PT:= T#200ms;
            SC_P2_StoperSrobovania.AlarmTime.PT:= T#10s;

            IF NOT TRCB_P2_Srobovanie_ST5.STATUS.KomunikaciaUkoncena THEN
                IF TRCB_P2_Srobovanie_ST5.OUTPUTS.PovolenieCinnostiNaPaletke = 'OK' THEN
                    SC_P2_StoperSrobovania.ResetStep:= TRUE;
                    SC_P2_StoperSrobovania.Step:= 555;
                ELSIF TRCB_P2_Srobovanie_ST5.OUTPUTS.PovolenieCinnostiNaPaletke = 'NG' THEN
                    Paletka[i].PAR.StavPaletky:= 'NG';
                    SC_P2_StoperSrobovania.ResetStep:= TRUE;
                    SC_P2_StoperSrobovania.Step:= 555;
                END_IF
            END_IF

        555:
            SC_P2_StoperSrobovania.StepName:='555 - Automaticky Rezim - vyhodnotenie stavu paletky';
            SC_P2_StoperSrobovania.IdleTime.PT:= T#200ms;
            SC_P2_StoperSrobovania.AlarmTime.PT:= T#10s;

            IF Paletka[i].PAR.StavPaletky = 'OK' THEN
                IF Paletka[i].PAR.StavPowerCP = 'PASS' THEN
                    Paletka[i].PAR.StavPaletky:= 'OK';
                ELSIF Paletka[i].PAR.StavPowerCP = 'FAIL' THEN
                    Paletka[i].PAR.StavPaletky:= 'NG';
                END_IF
            END_IF
            Paletka[i].VnutornyStav.KomunikaciaUzavreta:= TRUE;
            SC_P2_StoperSrobovania.ResetStep:= TRUE;
            SC_P2_StoperSrobovania.Step:= 560;

            //Vyvezenie paletky//

        560:
            SC_P2_StoperSrobovania.StepName:='560 - Automaticky Rezim - cakam na vyvezenie na stoper zvarania';
            SC_P2_StoperSrobovania.IdleTime.PT:= T#200ms;
            SC_P2_StoperSrobovania.AlarmTime.PT:= T#5s;

            P2_Robot.STAV.Srobovanie_PrebiehaManipulacia:= FALSE;

            IF P2_StoperSrobovania.KoniecCyklu THEN
                SC_P2_StoperSrobovania.ResetStep:= TRUE;
                SC_P2_StoperSrobovania.Step:= 0;
            ELSIF P2_StoperSrobovania.STAV.Porucha THEN
                Paletka[i].PAR.StavPaletky:= 'NG';
                P2_PoruchaST3:= TRUE;
            ELSIF ((NOT P2_StoperZvarania.IN.PritomnostPaletky_S9 AND SC_P2_StoperZvarania.Step = 100) OR (P2_StoperZvarania.OUT.ZasunStoper_YV59 AND SC_P2_StoperZvarania.Step = 561)) AND NOT P2_StoperSrobovania.STAV.PrebiehaVyvezeniePaletky THEN
                P2_StoperSrobovania.OUT.ZasunStoper_YV56:= TRUE;
                P2_StoperSrobovania.STAV.PrebiehaVyvezeniePaletky:= TRUE;
                SC_P2_StoperSrobovania.ResetStep:= TRUE;
                SC_P2_StoperSrobovania.Step:= 561;
            END_IF

        561:
            SC_P2_StoperSrobovania.StepName:='561 - Automaticky Rezim - ukoncenie vyvazania na stoper zvarania';
            SC_P2_StoperSrobovania.IdleTime.PT:= T#1300ms;
            SC_P2_StoperSrobovania.AlarmTime.PT:= T#10s;

            SC_P2_StoperSrobovania.AlarmTime.IN:= P2_StoperSrobovania.IN.PritomnostPaletky_S8;
            SC_P2_StoperSrobovania.IdleTime.IN:= NOT P2_StoperSrobovania.IN.PritomnostPaletky_S8;

            IF NOT P2_StoperSrobovania.IN.PritomnostPaletky_S8 THEN
                IF Revork THEN
                    Paletka[i].PAR.RevorkovyKus:= FALSE;
                    Paletka[i].PAR.CisloRevorkovejStanice:= '';
                    Revork:= FALSE;
                END_IF
                TestovaciKus:= FALSE;
                DoskrutkovaniePriPoruche:= FALSE;
                CisloFotky:= 0;
                Paletka[i].PAR.StavPowerCP:= '';
                Paletka[i].VnutornyStav.CinnostSpustena:= FALSE;
                Paletka[i].VnutornyStav.CinnostUkoncena:= FALSE;
                Paletka[i].VnutornyStav.FotkyOdoslane:= FALSE;
                Paletka[i].VnutornyStav.KomunikaciaOtvorena:= FALSE;
                Paletka[i].VnutornyStav.KomunikaciaUzavreta:= FALSE;
                Reports.Skrutkovacky.Moment_ToleranciaMIN.P2_LavaSkrutkaM6:= '';
                Reports.Skrutkovacky.Moment_ToleranciaMAX.P2_LavaSkrutkaM6:= '';
                Reports.Skrutkovacky.Moment_NameranaHodnota.P2_LavaSkrutkaM6:= '';
                Reports.Skrutkovacky.VyslednyReport.P2_LavaSkrutkaM6:= '';
                Reports.Skrutkovacky.Uhol_ToleranciaMIN.P2_LavaSkrutkaM6:= '';
                Reports.Skrutkovacky.Uhol_ToleranciaMAX.P2_LavaSkrutkaM6:= '';
                Reports.Skrutkovacky.Uhol_NameranaHodnota.P2_LavaSkrutkaM6:= '';
                Reports.Skrutkovacky.CasSkrutkovania.P2_LavaSkrutkaM6:= '';
                Reports.Skrutkovacky.VyskaSkrutkovania.P2_LavaSkrutkaM6:= '';
                Reports.Skrutkovacky.Moment_ToleranciaMIN.P2_PravaSkrutkaM6:= '';
                Reports.Skrutkovacky.Moment_ToleranciaMAX.P2_PravaSkrutkaM6:= '';
                Reports.Skrutkovacky.Moment_NameranaHodnota.P2_PravaSkrutkaM6:= '';
                Reports.Skrutkovacky.VyslednyReport.P2_PravaSkrutkaM6:= '';
                Reports.Skrutkovacky.Uhol_ToleranciaMIN.P2_PravaSkrutkaM6:= '';
                Reports.Skrutkovacky.Uhol_ToleranciaMAX.P2_PravaSkrutkaM6:= '';
                Reports.Skrutkovacky.Uhol_NameranaHodnota.P2_PravaSkrutkaM6:= '';
                Reports.Skrutkovacky.CasSkrutkovania.P2_PravaSkrutkaM6:= '';
                Reports.Skrutkovacky.VyskaSkrutkovania.P2_PravaSkrutkaM6:= '';
                Reports.Skrutkovacky.Moment_ToleranciaMIN.P2_LavaSkrutkaM4:= '';
                Reports.Skrutkovacky.Moment_ToleranciaMAX.P2_LavaSkrutkaM4:= '';
                Reports.Skrutkovacky.Moment_NameranaHodnota.P2_LavaSkrutkaM4:= '';
                Reports.Skrutkovacky.VyslednyReport.P2_LavaSkrutkaM4:= '';
                Reports.Skrutkovacky.Uhol_ToleranciaMIN.P2_LavaSkrutkaM4:= '';
                Reports.Skrutkovacky.Uhol_ToleranciaMAX.P2_LavaSkrutkaM4:= '';
                Reports.Skrutkovacky.Uhol_NameranaHodnota.P2_LavaSkrutkaM4:= '';
                Reports.Skrutkovacky.CasSkrutkovania.P2_LavaSkrutkaM4:= '';
                Reports.Skrutkovacky.VyskaSkrutkovania.P2_LavaSkrutkaM4:= '';
                Reports.Skrutkovacky.Moment_ToleranciaMIN.P2_PravaSkrutkaM4:= '';
                Reports.Skrutkovacky.Moment_ToleranciaMAX.P2_PravaSkrutkaM4:= '';
                Reports.Skrutkovacky.Moment_NameranaHodnota.P2_PravaSkrutkaM4:= '';
                Reports.Skrutkovacky.VyslednyReport.P2_PravaSkrutkaM4:= '';
                Reports.Skrutkovacky.Uhol_ToleranciaMIN.P2_PravaSkrutkaM4:= '';
                Reports.Skrutkovacky.Uhol_ToleranciaMAX.P2_PravaSkrutkaM4:= '';
                Reports.Skrutkovacky.Uhol_NameranaHodnota.P2_PravaSkrutkaM4:= '';
                Reports.Skrutkovacky.CasSkrutkovania.P2_PravaSkrutkaM4:= '';
                Reports.Skrutkovacky.VyskaSkrutkovania.P2_PravaSkrutkaM4:= '';
                Reports.Skrutkovacky.Moment_ToleranciaMIN.P2_LavaSkrutkaM5:= '';
                Reports.Skrutkovacky.Moment_ToleranciaMAX.P2_LavaSkrutkaM5:= '';
                Reports.Skrutkovacky.Moment_NameranaHodnota.P2_LavaSkrutkaM5:= '';
                Reports.Skrutkovacky.VyslednyReport.P2_LavaSkrutkaM5:= '';
                Reports.Skrutkovacky.Uhol_ToleranciaMIN.P2_LavaSkrutkaM5:= '';
                Reports.Skrutkovacky.Uhol_ToleranciaMAX.P2_LavaSkrutkaM5:= '';
                Reports.Skrutkovacky.Uhol_NameranaHodnota.P2_LavaSkrutkaM5:= '';
                Reports.Skrutkovacky.CasSkrutkovania.P2_LavaSkrutkaM5:= '';
                Reports.Skrutkovacky.VyskaSkrutkovania.P2_LavaSkrutkaM5:= '';
                Reports.Skrutkovacky.Moment_ToleranciaMIN.P2_PravaSkrutkaM5:= '';
                Reports.Skrutkovacky.Moment_ToleranciaMAX.P2_PravaSkrutkaM5:= '';
                Reports.Skrutkovacky.Moment_NameranaHodnota.P2_PravaSkrutkaM5:= '';
                Reports.Skrutkovacky.VyslednyReport.P2_PravaSkrutkaM5:= '';
                Reports.Skrutkovacky.Uhol_ToleranciaMIN.P2_PravaSkrutkaM5:= '';
                Reports.Skrutkovacky.Uhol_ToleranciaMAX.P2_PravaSkrutkaM5:= '';
                Reports.Skrutkovacky.Uhol_NameranaHodnota.P2_PravaSkrutkaM5:= '';
                Reports.Skrutkovacky.CasSkrutkovania.P2_PravaSkrutkaM5:= '';
                Reports.Skrutkovacky.VyskaSkrutkovania.P2_PravaSkrutkaM5:= '';
                Reports.Skrutkovacky.Moment_ToleranciaMIN.P2_StrednaSkrutkaM4:= '';
                Reports.Skrutkovacky.Moment_ToleranciaMAX.P2_StrednaSkrutkaM4:= '';
                Reports.Skrutkovacky.Moment_NameranaHodnota.P2_StrednaSkrutkaM4:= '';
                Reports.Skrutkovacky.VyslednyReport.P2_StrednaSkrutkaM4:= '';
                Reports.Skrutkovacky.Uhol_ToleranciaMIN.P2_StrednaSkrutkaM4:= '';
                Reports.Skrutkovacky.Uhol_ToleranciaMAX.P2_StrednaSkrutkaM4:= '';
                Reports.Skrutkovacky.Uhol_NameranaHodnota.P2_StrednaSkrutkaM4:= '';
                Reports.Skrutkovacky.CasSkrutkovania.P2_StrednaSkrutkaM4:= '';
                Reports.Skrutkovacky.VyskaSkrutkovania.P2_StrednaSkrutkaM4:= '';
                Reports.Kamery.P2_CAM10_KontrolaPaletky:= '';
                P2_Srobov_ManipulaciaUkoncena:= FALSE;
            END_IF

            IF SC_P2_StoperSrobovania.IdleTime.Q  THEN
                P2_StoperSrobovania.OUT.ZasunStoper_YV56:= FALSE;
                SC_P2_StoperSrobovania.ResetStep:= TRUE;
                SC_P2_StoperSrobovania.Step:= 100;
            ELSIF SC_P2_StoperSrobovania.AlarmTime.Q THEN
                P2_Alarmy[288]:= TRUE;
                P2_Pracovisko.KoniecCyklu:= TRUE;
                SC_P2_StoperSrobovania.ResetStep:= TRUE;
                SC_P2_StoperSrobovania.Step:= 0;
            END_IF

            //*******************************************************Manuálny režim*******************************************************************************//

        700:
            SC_P2_StoperSrobovania.StepName:='700 - Manualny Rezim';
            SC_P2_StoperSrobovania.IdleTime.PT:= T#8s;
            SC_P2_StoperSrobovania.AlarmTime.PT:= T#5s;

    END_CASE

				END_PROGRAM

PROGRAM _EXIT
				(* Insert code here *)

				END_PROGRAM
```

#### Variables.var - Local variables
```iecst
VAR
	SC_OvlCentrovacky : SequenceControlTyp;
	Centrovacku_VYSUN : BOOL;
	Centrovacku_ZASUN : BOOL;
	PrecitaneCisloPaletky : STRING[3];
	ServerOdpoved_StavPowerCP : STRING[5];
	i : USINT;
	TEST : BOOL;
	PocetDopytovNaServer : USINT;
	TestovaciKus : BOOL;
	Revork : BOOL;
	Triger_0 : BOOL;
	Triger_1 : BOOL;
	CisloFotky : USINT;
	Round_0 : Round;
	Round_1 : Round;
	Round_2 : Round;
	a : USINT;
	VysunutieSkrutkovacky_OK : BOOL;
	PocetTrigrovKamery : USINT;
	DoskrutkovaniePriPoruche : BOOL;
END_VAR
```

#### OvlCentrovacky.st
```iecst
ACTION OvlCentrovacky:

	//Volanie funkcie SequenceControl//
	SequenceControl(SC:= SC_OvlCentrovacky);

	CASE SC_OvlCentrovacky.Step OF

		0:
			SC_OvlCentrovacky.StepName:= '0 - Nulovanie';
			Centrovacku_VYSUN:= FALSE;
			Centrovacku_ZASUN:= FALSE;
//			P2_StoperSrobovania.OUT.VysunCentrovanie_YV57:= FALSE;
//			P2_StoperSrobovania.OUT.ZasunCentrovanie_YV58:= FALSE;

			IF SC_P2_StoperSrobovania.Step <> 0 THEN
				SC_OvlCentrovacky.ResetStep:= TRUE;
				SC_OvlCentrovacky.Step:= 1;
			END_IF

		1:
			SC_OvlCentrovacky.StepName:= '1 - Rozhodnutie o cinnosti';
			IF Centrovacku_VYSUN THEN
				SC_OvlCentrovacky.Step:= 10;
			ELSIF Centrovacku_ZASUN THEN
				SC_OvlCentrovacky.Step:= 20;
			END_IF

		10:
			SC_OvlCentrovacky.StepName:= '10 - Vysunutie centrovacky';
			SC_OvlCentrovacky.IdleTime.PT:= T#3s;
			SC_OvlCentrovacky.AlarmTime.PT:= T#3s;

			IF P2_StoperSrobovania.Automat THEN
				SC_OvlCentrovacky.AlarmTime.IN:= TRUE;
			ELSE
				SC_OvlCentrovacky.IdleTime.IN:= TRUE;
			END_IF

			IF NOT SC_OvlCentrovacky.Switch1 THEN
				P2_StoperSrobovania.OUT.ZasunCentrovanie_YV58:= FALSE;
                P2_StoperSrobovania.OUT.VysunCentrovanie_YV57:= TRUE;
				SC_OvlCentrovacky.Switch1:= TRUE;
			END_IF

			IF P2_StoperSrobovania.IN.Centrovanie_VYSUNUTE_IS14 OR SC_OvlCentrovacky.IdleTime.Q THEN
				SC_OvlCentrovacky.ResetStep:= TRUE;
				SC_OvlCentrovacky.Step:= 0;
			ELSIF SC_OvlCentrovacky.AlarmTime.Q THEN
				P2_Alarmy[212]:= TRUE;
				P2_PoruchaST2:= TRUE;
			END_IF

		20:
			SC_OvlCentrovacky.StepName:= '20 - Zasunutie centrovacky';
			SC_OvlCentrovacky.IdleTime.PT:= T#3s;
			SC_OvlCentrovacky.AlarmTime.PT:= T#3s;

			IF P2_StoperSrobovania.Automat THEN
				SC_OvlCentrovacky.AlarmTime.IN:= TRUE;
			ELSE
				SC_OvlCentrovacky.IdleTime.IN:= TRUE;
			END_IF

			IF NOT SC_OvlCentrovacky.Switch1 THEN
				P2_StoperSrobovania.OUT.VysunCentrovanie_YV57:= FALSE;
                P2_StoperSrobovania.OUT.ZasunCentrovanie_YV58:= TRUE;
				SC_OvlCentrovacky.Switch1:= TRUE;
			END_IF

			IF P2_StoperSrobovania.IN.Centrovanie_ZASUNUTE_IS15 OR SC_OvlCentrovacky.IdleTime.Q THEN
				SC_OvlCentrovacky.ResetStep:= TRUE;
				SC_OvlCentrovacky.Step:= 0;
			ELSIF SC_OvlCentrovacky.AlarmTime.Q THEN
				P2_Alarmy[213]:= TRUE;
				P2_PoruchaST2:= TRUE;
			END_IF

	END_CASE

END_ACTION
```

#### StratoveSekundy.st
```iecst
ACTION StratoveSekundy:

END_ACTION
```

#### IOLinkKomunikacia.st
```iecst
ACTION IOLinkKomunikacia:

	//Snímač paletky//
	P2_StoperSrobovania.IN.PritomnostPaletky_S8:= P2_StoperSrobovania.PAR.SnimacPaletky_IOLinkInputs[1].0;
	P2_StoperSrobovania.IN.PrecitaneCisloPaletky_S8:= P2_StoperSrobovania.PAR.SnimacPaletky_IOLinkInputs[9];

    //Snímač vysunutia šrobovačky M4//
    Round_0.VstupnaHodnota:= P2_Srobovanie.IN.SkrutkM4_VysunutieHrotu_IOlink;
    P2_Srobovanie.IN.SkrutkM4_VysunutieHrotu_IOS4:= Round_0.VystupnaHodnota;
    Round_0();

    //Snímač vysunutia šrobovačky M5//
    Round_1.VstupnaHodnota:= P2_Srobovanie.IN.SkrutkM5_VysunutieHrotu_IOlink;
    P2_Srobovanie.IN.SkrutkM5_VysunutieHrotu_IOS5:= Round_1.VystupnaHodnota;
    Round_1();

    //Snímač vysunutia šrobovačky M6//
    Round_2.VstupnaHodnota:= P2_Srobovanie.IN.SkrutkM6_VysunutieHrotu_IOlink;
    P2_Srobovanie.IN.SkrutkM6_VysunutieHrotu_IOS3:= Round_2.VystupnaHodnota;
    Round_2();

END_ACTION
```

### Program Logical/Program/Pracovisko_2/P2_Srobovanie (IEC)
